Staubli VAL3: RobotCommand.dtx

public bool bIsValid = false
public num nMode
public num nRemoteCtrlPeriod
public num nMotionCmdType
public num nMotionCmdData[6]
public bool nDigitalOutputs[16]
public num nAnalogOutputs[4]
